(* Schneider Machine Expert - Basic project New project, file version 2.6.0.0 *)
(* CompanyInformations: Name=PT. SIIX ELECTRONICS INDONESIA *)
(* ProjectInformations: Name=AUTOMATIC LEAD CUTTING FORMING *)

HARDWARE
  Cpu 0: TM221CE40R
  EthernetConfiguration: NetworkName=M221, IpAllocationMode=FixedAddress, IpAddress=192.168.0.2, SubnetMask=255.255.255.0
  SerialLineConfiguration: Baud=Baud19200, Parity=ParityEven, DataBits=DataBits8, StopBits=StopBits1, PhysicalMedium=PhysicalMediumRs485, TransmissionMode=TransmissionModeModbusRtu, SlaveId=1, Addressing=SlaveAddressing
  MastTask: UsePeriodScanMode=false, PeriodScan=100
  FastTask: Period=255
  CpuBehavior: StartingMode=StartAsPreviousState, AutoSaveRamOnEeprom=true, WatchdogPeriod=250

SYMBOLS  (address, symbol, comment, settings)
  %M0         "POLARITY RESULT"
  %M1         "RORO"
  %M2         "GRIPPER OFF"
  %M4         "PROG START"
  %I0.0       "EMERGENCY"
  %I0.1       "BTN START"
  %I0.2       "SENSOR R CUT FWD"
  %I0.3       "SENSOR R CUT BCK"
  %I0.4       "SENSOR L CUT FWD"
  %I0.5       "SENSOR L CUT BCK"
  %I0.6       "ROTATE CW"
  %I0.7       "ROTATE CCW"
  %I0.8       "GRIPPER TRF COMP OFF"
  %I0.9       "ROTATE GRIP CLOSE"
  %I0.10      "GRIPPER TRF COMP OFF"
  %I0.11      "COMP GRIPPER CLOSE"
  %I0.12      "SENSOR TRF FWD"
  %I0.13      "SENSOR TRF BCK"
  %I0.14      "PART DETECTION"
  %I0.15      "POLARITY CHECK"
  %Q0.0       "R CUT"
  %Q0.1       "L CUT"
  %Q0.2       "ROTATE PART"
  %Q0.3       "ROTATE GRIP"
  %Q0.4       "GRIPPER TRF COMP"
  %Q0.5       "COMP TRANSFER FWD"
  %Q0.6       "BOWLFEEDER"
  %Q0.7       "POLARITY RESULT"
  %Q0.9       "RORO"
  %Q0.11      "TL-RED"
  %Q0.13      "TL-GREEN"

POU New POU
  (* SectionNumber=1 *)

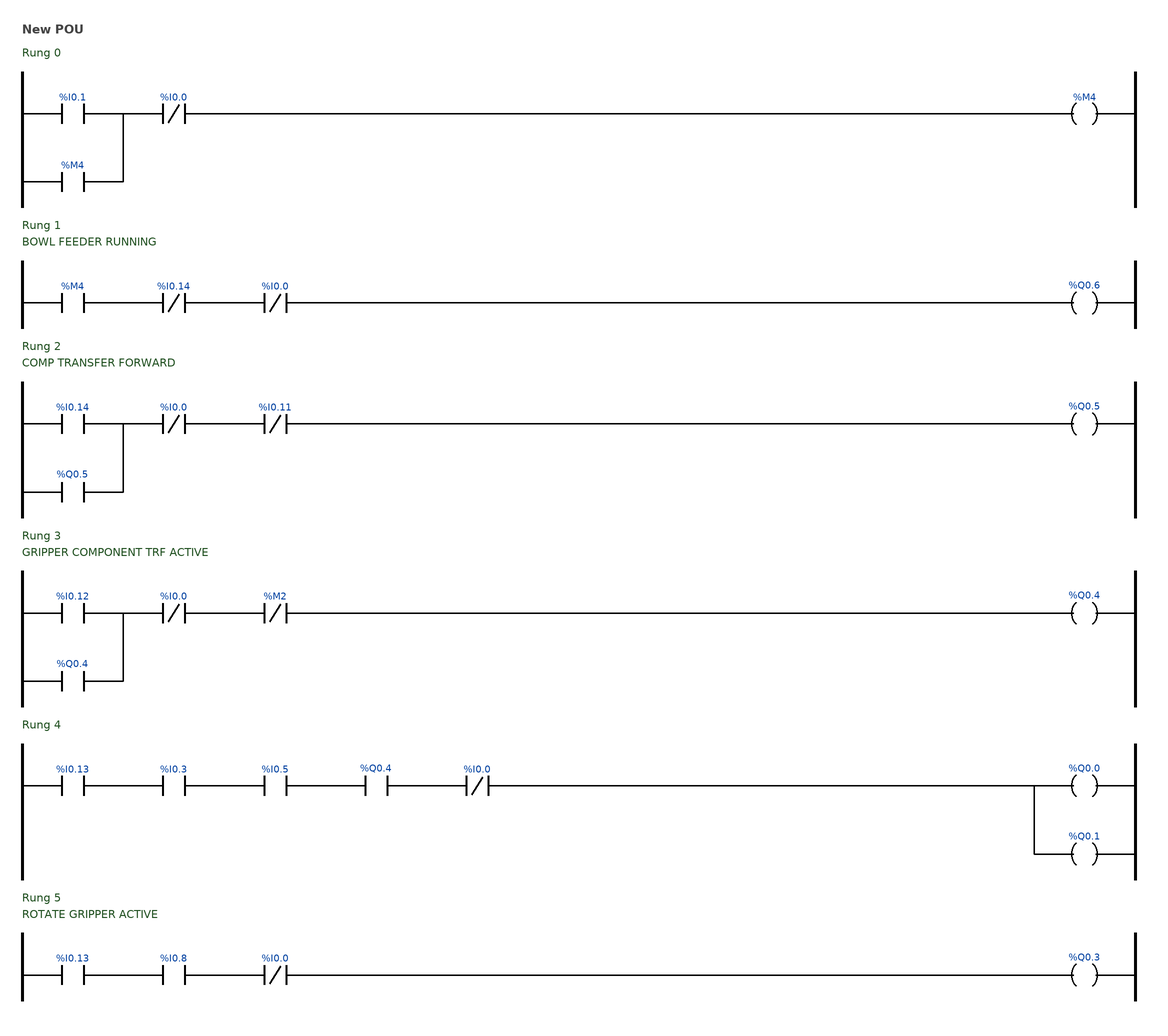

// Rung 0
  LD %I0.1
  OR %M4
  ANDN %I0.0
  ST %M4
  // as ST:
  //   %M4 := (%I0.1 OR %M4) AND NOT %I0.0;

// Rung 1
// BOWL FEEDER RUNNING
  LD %M4
  ANDN %I0.14
  ANDN %I0.0
  ST %Q0.6
  // as ST:
  //   %Q0.6 := %M4 AND NOT %I0.14 AND NOT %I0.0;

// Rung 2
// COMP TRANSFER FORWARD
  LD %I0.14
  OR %Q0.5
  ANDN %I0.0
  ANDN %I0.11
  ST %Q0.5
  // as ST:
  //   %Q0.5 := (%I0.14 OR %Q0.5) AND NOT %I0.0 AND NOT %I0.11;

// Rung 3
// GRIPPER COMPONENT TRF ACTIVE
  LD %I0.12
  OR %Q0.4
  ANDN %I0.0
  ANDN %M2
  ST %Q0.4
  // as ST:
  //   %Q0.4 := (%I0.12 OR %Q0.4) AND NOT %I0.0 AND NOT %M2;

// Rung 4
  LD %I0.13
  AND %I0.3
  AND %I0.5
  AND %Q0.4
  ANDN %I0.0
  ST %Q0.0
  ST %Q0.1
  // as ST:
  //   %Q0.0 := %I0.13 AND %I0.3 AND %I0.5 AND %Q0.4 AND NOT %I0.0;
  //   %Q0.1 := %I0.13 AND %I0.3 AND %I0.5 AND %Q0.4 AND NOT %I0.0;

// Rung 5
// ROTATE GRIPPER ACTIVE
  LD %I0.13
  AND %I0.8
  ANDN %I0.0
  ST %Q0.3
  // as ST:
  //   %Q0.3 := %I0.13 AND %I0.8 AND NOT %I0.0;

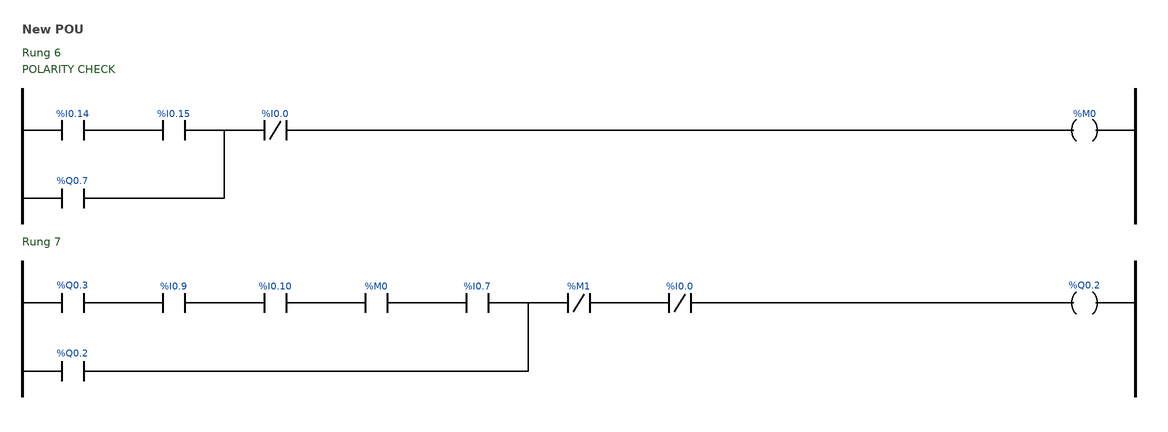

// Rung 6
// POLARITY CHECK
  LD %I0.14
  AND %I0.15
  OR %Q0.7
  ANDN %I0.0
  ST %M0
  // as ST:
  //   %M0 := (%I0.14 AND %I0.15 OR %Q0.7) AND NOT %I0.0;

// Rung 7
  LD %Q0.3
  AND %I0.9
  AND %I0.10
  AND %M0
  AND %I0.7
  OR %Q0.2
  ANDN %M1
  ANDN %I0.0
  ST %Q0.2
  // as ST:
  //   %Q0.2 := (%Q0.3 AND %I0.9 AND %I0.10 AND %M0 AND %I0.7 OR %Q0.2) AND NOT %M1 AND NOT %I0.0;
